// TIA Portal project "babu_schoolBell" (V15)

(* hardware
DEVICE "S7-1200 station_1"  S7-1200 Station
   slot 0: "Rack_0"  S7-1200 Rack  Rack  V1.0
   slot 1: "PLC_1"  CPU 1212C DC/DC/DC  6ES7 212-1AE40-0XB0  V4.2
*)

// ===== PLC "PLC_1"  CPU 1212C DC/DC/DC =====

VAR_GLOBAL   // PLC tag table "Default tag table"
   "POWER ON" AT %M0.0 : Bool;
   "OUTPUT" AT %Q0.0 : Bool;
   "MEMORY" AT %M0.1 : Bool;
   "TEST" AT %M0.2 : Bool;
   "RING BELL" AT %Q0.1 : Bool;
   "RING BELL MEMORY" AT %M0.3 : Bool;
   "TIMER POWER ON" AT %M0.4 : Bool;
   "TIMER OUTPUT" AT %Q0.2 : Bool;
   "TIMER LOW OUTPUT" AT %M0.5 : Bool;
   "TIMER POWER ON 1" AT %M0.6 : Bool;
   "TIMER OUTPUT 1" AT %Q0.3 : Bool;
   "TIMER MEMORY 1" AT %M0.7 : Bool;
   "POWER ON TONR" AT %M1.0 : Bool;
   "TONR OUTPUT" AT %M1.1 : Bool;
   "DELAY PUSH BUTTON" AT %M1.2 : Bool;
   "DELAY MEMORY" AT %M1.3 : Bool;
END_VAR

// folder: System blocks/Program resources

DATA_BLOCK "IEC_Timer_0_DB"   // DB1
{ S7_Optimized_Access := 'TRUE' }
AUTHOR : Simatic
FAMILY : IEC
NAME : IEC_TMR
VERSION : 1.0
// stored: InstanceOfName IEC_TIMER
"IEC_TIMER"
BEGIN
END_DATA_BLOCK

DATA_BLOCK "IEC_Timer_0_DB_4"   // DB5
{ S7_Optimized_Access := 'TRUE' }
AUTHOR : Simatic
FAMILY : IEC
NAME : IEC_TMR
VERSION : 1.0
// stored: InstanceOfName IEC_TIMER
"IEC_TIMER"
BEGIN
END_DATA_BLOCK

DATA_BLOCK "IEC_Timer_0_DB_5"   // DB6
{ S7_Optimized_Access := 'TRUE' }
AUTHOR : Simatic
FAMILY : IEC
NAME : IEC_TMR
VERSION : 1.0
// stored: InstanceOfName IEC_TIMER
"IEC_TIMER"
BEGIN
END_DATA_BLOCK

DATA_BLOCK "IEC_Timer_0_DB_6"   // DB7
{ S7_Optimized_Access := 'TRUE' }
AUTHOR : Simatic
FAMILY : IEC
NAME : IEC_TMR
VERSION : 1.0
// stored: InstanceOfName IEC_TIMER
"IEC_TIMER"
BEGIN
END_DATA_BLOCK

DATA_BLOCK "IEC_Timer_0_DB_7"   // DB8
{ S7_Optimized_Access := 'TRUE' }
AUTHOR : Simatic
FAMILY : IEC
NAME : IEC_TMR
VERSION : 1.0
// stored: InstanceOfName IEC_TIMER
"IEC_TIMER"
BEGIN
END_DATA_BLOCK

DATA_BLOCK "IEC_Timer_0_DB_8"   // DB9
{ S7_Optimized_Access := 'TRUE' }
AUTHOR : Simatic
FAMILY : IEC
NAME : IEC_TMR
VERSION : 1.0
// stored: InstanceOfName IEC_TIMER
"IEC_TIMER"
BEGIN
END_DATA_BLOCK

DATA_BLOCK "IEC_Timer_0_DB_9"   // DB10
{ S7_Optimized_Access := 'TRUE' }
AUTHOR : Simatic
FAMILY : IEC
NAME : IEC_TMR
VERSION : 1.0
// stored: InstanceOfName IEC_TIMER
"IEC_TIMER"
BEGIN
END_DATA_BLOCK

DATA_BLOCK "IEC_Timer_0_DB_10"   // DB11
{ S7_Optimized_Access := 'TRUE' }
AUTHOR : Simatic
FAMILY : IEC
NAME : IEC_TMR
VERSION : 1.0
// stored: InstanceOfName IEC_TIMER
"IEC_TIMER"
BEGIN
END_DATA_BLOCK

// folder: (top level)

ORGANIZATION_BLOCK "Main"   // OB1, LAD, ProgramCycle
TITLE = "Main Program Sweep (Cycle)"
{ S7_Optimized_Access := 'TRUE' }
VERSION : 0.1
   VAR_INPUT
      Initial_Call : Bool;   // Initial call of this OB
      Remanence : Bool;   // =True, if remanent data are available
   END_VAR
BEGIN

REGION Network 1
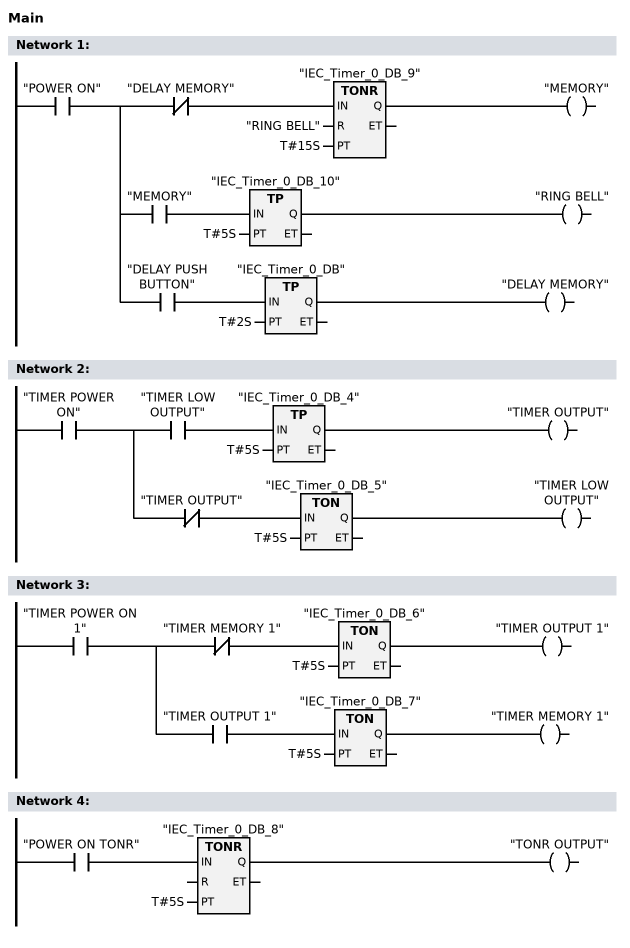
   "IEC_Timer_0_DB_9".TONR(IN := "POWER ON" AND NOT "DELAY MEMORY", R := "RING BELL", PT := T#15S);
   "MEMORY" := "IEC_Timer_0_DB_9".Q;
   "IEC_Timer_0_DB_10".TP(IN := "POWER ON" AND "MEMORY", PT := T#5S);
   "RING BELL" := "IEC_Timer_0_DB_10".Q;
   "IEC_Timer_0_DB".TP(IN := "POWER ON" AND "DELAY PUSH BUTTON", PT := T#2S);
   "DELAY MEMORY" := "IEC_Timer_0_DB".Q;
END_REGION

REGION Network 2
   "IEC_Timer_0_DB_4".TP(IN := "TIMER POWER ON" AND "TIMER LOW OUTPUT", PT := T#5S);
   "TIMER OUTPUT" := "IEC_Timer_0_DB_4".Q;
   "IEC_Timer_0_DB_5".TON(IN := "TIMER POWER ON" AND NOT "TIMER OUTPUT", PT := T#5S);
   "TIMER LOW OUTPUT" := "IEC_Timer_0_DB_5".Q;
END_REGION

REGION Network 3
   "IEC_Timer_0_DB_6".TON(IN := "TIMER POWER ON 1" AND NOT "TIMER MEMORY 1", PT := T#5S);
   "TIMER OUTPUT 1" := "IEC_Timer_0_DB_6".Q;
   "IEC_Timer_0_DB_7".TON(IN := "TIMER POWER ON 1" AND "TIMER OUTPUT 1", PT := T#5S);
   "TIMER MEMORY 1" := "IEC_Timer_0_DB_7".Q;
END_REGION

REGION Network 4
   "IEC_Timer_0_DB_8".TONR(IN := "POWER ON TONR", PT := T#5S);
   "TONR OUTPUT" := "IEC_Timer_0_DB_8".Q;
END_REGION
END_ORGANIZATION_BLOCK